KUKA KRL program: wkz6_off_st600.src, wkz6_off_st600.dat

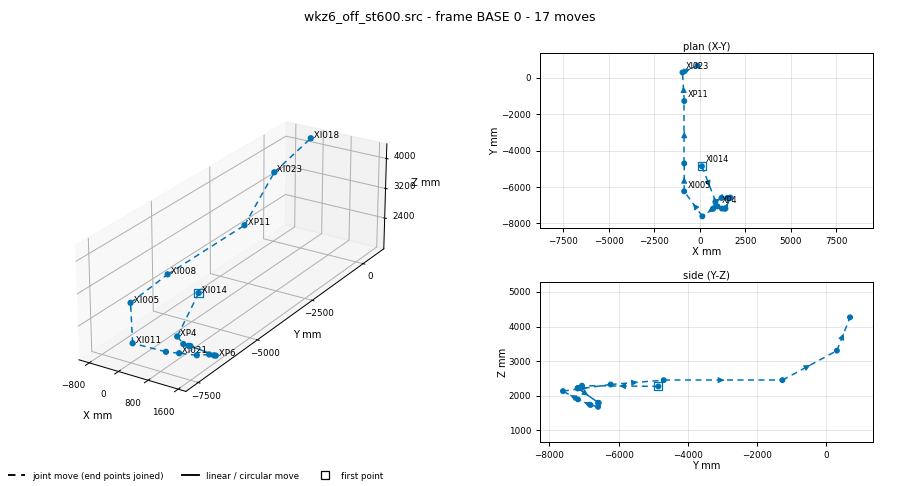
[picture p0: tool path of wkz6_off_st600.src in frame BASE 0, 17 of 17 moves have a stored position in this frame; points joined in program order, loops and branches not executed]
--- wkz6_off_st600.src ---
&ACCESS RVO4
&REL 118
&COMMENT Pega GRP AXOR GeoBox
&PARAM DISKPATH = KRC:\R1\Program\olp
&PARAM TEMPLATE = C:\KRC\Roboter\Template\vorgabe
&PARAM EDITMASK = *
DEF wkz6_off_st600( )
;FOLD INI
  ;FOLD BASISTECH INI
    GLOBAL INTERRUPT DECL 3 WHEN $STOPMESS==TRUE DO IR_STOPM ( )
    INTERRUPT ON 3
    BAS (#INITMOV,0)
  ;ENDFOLD (BASISTECH INI)
;FOLD GRIPPERTECH INI
USER_GRP(0,DUMMY,DUMMY,GDEFAULT)
;ENDFOLD (GRIPPERTECH INI)
  ;FOLD USER INI
    ;Make your modifications here

  ;ENDFOLD (USER INI)
;ENDFOLD (INI)

; Caracterizacao dos meios de producao
; Changes: Pega Gripper Axor na GeoBox
; Versao Atual: 20/08/2015
; Name: P13.050-R3

chk_w8_wechs_ok ( )   ; CHECK TOOL CHANGE

;FOLD ; Ponto Externo 7;%{PE}%R 8.2.20,%MKUKATPBASIS,%CCOMMENT,%VNORMAL,%P 2:Ponto Externo 7
;ENDFOLD
;FOLD PTP l014 Vel=100 % P_OLP34 Tool[8]:Tool Changer Base[0];%{PE}%R 8.2.20,%MKUKATPBASIS,%CMOVE,%VPTP,%P 1:PTP, 2:l014, 3:, 5:100, 7:P_OLP34
$BWDSTART=FALSE
PDAT_ACT=PP_OLP34
FDAT_ACT=Fl014
BAS(#PTP_PARAMS,100)
PTP Xl014
;ENDFOLD

; AGUARDA LIBERACAO PARA SAIR COM GARRA
;FOLD OUT 3378 'Lib. p/ retirar Gripper GeoBox' State=TRUE ;%{PE}%R 8.2.20,%MKUKATPBASIS,%COUT,%VOUTX,%P 2:3378, 3:Lib. p/ retirar Gripper GeoBox, 5:TRUE, 6:
$OUT[3378]=TRUE
;ENDFOLD
;FOLD WAIT FOR ( IN 3378 'Lib. p/ retirar Gripper GeoBox' );%{PE}%R 8.2.20,%MKUKATPBASIS,%CEXT_WAIT_FOR,%VEXT_WAIT_FOR,%P 2:, 4:, 5:$IN, 6:3378, 7:Lib. p/ retirar Gripper GeoBox, 9:
WAIT FOR  ( $IN[3378] )
;ENDFOLD
;FOLD OUT 3378 'Lib. p/ retirar Gripper GeoBox' State=FALSE ;%{PE}%R 8.2.20,%MKUKATPBASIS,%COUT,%VOUTX,%P 2:3378, 3:Lib. p/ retirar Gripper GeoBox, 5:FALSE, 6:
$OUT[3378]=FALSE
;ENDFOLD
;FOLD OUT 3348 'Fora area GEOBOX' State=FALSE ;%{PE}%R 8.2.20,%MKUKATPBASIS,%COUT,%VOUTX,%P 2:3348, 3:Fora area GEOBOX, 5:FALSE, 6:
$OUT[3348]=FALSE
;ENDFOLD

; LIGA INTERTRAVAMENTO 1 C/ R1 GARRA
;FOLD Collision.Monitoring_1_On ;%{PE}%MKUKATPUSER
COLLSTOP( 1, 1 ) ;Interrupt-Controlled
;ENDFOLD

; LIGA INTERTRAVAMENTO 5 C/ R5 GARRA
;FOLD Collision.Monitoring_5_On ;%{PE}%MKUKATPUSER
COLLSTOP( 5, 1 ) ;not Interrupt-Controlled
;ENDFOLD

;FOLD PTP P4 CONT Vel=100 % PDAT2 Tool[6]:Gripper G0100R Base[0];%{PE}%R 8.2.20,%MKUKATPBASIS,%CMOVE,%VPTP,%P 1:PTP, 2:P4, 3:C_DIS, 5:100, 7:PDAT2
$BWDSTART=FALSE
PDAT_ACT=PPDAT2
FDAT_ACT=FP4
BAS(#PTP_PARAMS,100)
PTP XP4 C_DIS
;ENDFOLD
;FOLD PTP P7 CONT Vel=100 % PDAT3 Tool[6]:Gripper G0100R Base[0];%{PE}%R 8.2.20,%MKUKATPBASIS,%CMOVE,%VPTP,%P 1:PTP, 2:P7, 3:C_DIS, 5:100, 7:PDAT3
$BWDSTART=FALSE
PDAT_ACT=PPDAT3
FDAT_ACT=FP7
BAS(#PTP_PARAMS,100)
PTP XP7 C_DIS
;ENDFOLD
;FOLD LIN l041 Vel=0.25 m/s L_OLP3 Tool[8]:Tool Changer Base[0];%{PE}%R 8.2.20,%MKUKATPBASIS,%CMOVE,%VLIN,%P 1:LIN, 2:l041, 3:, 5:0.25, 7:L_OLP3
$BWDSTART=FALSE
LDAT_ACT=LL_OLP3
FDAT_ACT=Fl041
BAS(#CP_PARAMS,0.25)
LIN Xl041
;ENDFOLD

; AGUARDA MPS DESTRAVADO
;FOLD OUT 224 'Bloquear MPS' State=FALSE ;%{PE}%R 8.2.20,%MKUKATPBASIS,%COUT,%VOUTX,%P 2:224, 3:Bloquear MPS, 5:FALSE, 6:
$OUT[224]=FALSE
;ENDFOLD
;FOLD OUT 223 'Desbloquear MPS' State=TRUE ;%{PE}%R 8.2.20,%MKUKATPBASIS,%COUT,%VOUTX,%P 2:223, 3:Desbloquear MPS, 5:TRUE, 6:
$OUT[223]=TRUE
;ENDFOLD
;FOLD WAIT FOR ( IN 217 'MPS Destravado' );%{PE}%R 8.2.20,%MKUKATPBASIS,%CEXT_WAIT_FOR,%VEXT_WAIT_FOR,%P 2:, 4:, 5:$IN, 6:217, 7:MPS Destravado, 9:
WAIT FOR  ( $IN[217] )
;ENDFOLD
;FOLD WAIT FOR NOT ( IN 221 'MPS Travado' );%{PE}%R 8.2.20,%MKUKATPBASIS,%CEXT_WAIT_FOR,%VEXT_WAIT_FOR,%P 2:NOT, 4:, 5:$IN, 6:221, 7:MPS Travado, 9:
WAIT FOR  NOT ( $IN[221] )
;ENDFOLD

;FOLD ; Posicao de Pega Gripper AXOR na GeoBox;%{PE}%R 8.2.20,%MKUKATPBASIS,%CCOMMENT,%VNORMAL,%P 2:Posicao de Pega Gripper AXOR  na  GeoBox
;ENDFOLD
;FOLD LIN P_DE11 Vel=0.25 m/s L_OLP4 Tool[8]:Tool Changer Base[0];%{PE}%R 8.2.20,%MKUKATPBASIS,%CMOVE,%VLIN,%P 1:LIN, 2:P_DE11, 3:, 5:0.25, 7:L_OLP4
$BWDSTART=FALSE
LDAT_ACT=LL_OLP4
FDAT_ACT=FP_DE11
BAS(#CP_PARAMS,0.25)
LIN XP_DE11
;ENDFOLD

;FOLD OUT 3379 'Lib. p/ sair c/ Gripper GeoBox' State=TRUE ;%{PE}%R 8.2.20,%MKUKATPBASIS,%COUT,%VOUTX,%P 2:3379, 3:Lib. p/ sair c/ Gripper GeoBox, 5:TRUE, 6:
$OUT[3379]=TRUE
;ENDFOLD

;FOLD WAIT FOR ( IN 219 'Posicao p/ Acoplamento OK' );%{PE}%R 8.2.20,%MKUKATPBASIS,%CEXT_WAIT_FOR,%VEXT_WAIT_FOR,%P 2:, 4:, 5:$IN, 6:219, 7:Posicao p/ Acoplamento OK, 9:
WAIT FOR  ( $IN[219] )
;ENDFOLD
;FOLD WAIT Time=0.5 sec;%{PE}%R 8.2.20,%MKUKATPBASIS,%CWAIT,%VWAIT,%P 3:0.5
WAIT SEC 0.5
;ENDFOLD
;FOLD OUT 223 'Desbloquear MPS' State=FALSE ;%{PE}%R 8.2.20,%MKUKATPBASIS,%COUT,%VOUTX,%P 2:223, 3:Desbloquear MPS, 5:FALSE, 6:
$OUT[223]=FALSE
;ENDFOLD
;FOLD OUT 224 'Bloquear MPS' State=TRUE ;%{PE}%R 8.2.20,%MKUKATPBASIS,%COUT,%VOUTX,%P 2:224, 3:Bloquear MPS, 5:TRUE, 6:
$OUT[224]=TRUE
;ENDFOLD
;FOLD WAIT FOR NOT ( IN 217 'MPS Destravado' );%{PE}%R 8.2.20,%MKUKATPBASIS,%CEXT_WAIT_FOR,%VEXT_WAIT_FOR,%P 2:NOT, 4:, 5:$IN, 6:217, 7:MPS Destravado, 9:
WAIT FOR  NOT ( $IN[217] )
;ENDFOLD
;FOLD WAIT FOR ( IN 221 'MPS Travado' );%{PE}%R 8.2.20,%MKUKATPBASIS,%CEXT_WAIT_FOR,%VEXT_WAIT_FOR,%P 2:, 4:, 5:$IN, 6:221, 7:MPS Travado, 9:
WAIT FOR  ( $IN[221] )
;ENDFOLD
;FOLD IBUS ON SEGMENT_4;%{PE}%R 8.2.20,%MKUKATPBASIS,%CIBUS,%VMAP,%P 2:#ON, 3:4
$IBUS_ON=IBUS_SEGMENT[4]
$IBUS_OFF=0
;ENDFOLD
;FOLD WAIT Time=0.5 sec;%{PE}%R 8.2.20,%MKUKATPBASIS,%CWAIT,%VWAIT,%P 3:0.5
WAIT SEC 0.5
;ENDFOLD

; ABRE GRAMPOS
;FOLD SET Z2.1 RPS AXOR State=OPN GDAT15;%{PE}%R 8.2.1,%MKUKATPGRP,%CGRP,%VGRP,%P 2:10, 4:1, 5:#NO, 6:GDAT15, 8:0, 10:0
H50(GRP,10,1,GGDAT15)
;ENDFOLD
;FOLD SET Z4.1 GRP AXOR State=OPN GDAT12;%{PE}%R 8.2.1,%MKUKATPGRP,%CGRP,%VGRP,%P 2:12, 4:1, 5:#NO, 6:GDAT12, 8:0, 10:0
H50(GRP,12,1,GGDAT12)
;ENDFOLD
;FOLD SET Z5.1/2/3/4 GRP AXOR State=OPN GDAT16;%{PE}%R 8.2.1,%MKUKATPGRP,%CGRP,%VGRP,%P 2:13, 4:1, 5:#NO, 6:GDAT16, 8:0, 10:0
H50(GRP,13,1,GGDAT16)
;ENDFOLD
;FOLD SET Z6.1/2/3/4 GRP AXOR State=OPN GDAT17;%{PE}%R 8.2.1,%MKUKATPGRP,%CGRP,%VGRP,%P 2:14, 4:1, 5:#NO, 6:GDAT17, 8:0, 10:0
H50(GRP,14,1,GGDAT17)
;ENDFOLD
;FOLD SET Z7.1/2 GRP AXOR State=OPN GDAT18;%{PE}%R 8.2.1,%MKUKATPGRP,%CGRP,%VGRP,%P 2:15, 4:1, 5:#NO, 6:GDAT18, 8:0, 10:0
H50(GRP,15,1,GGDAT18)
;ENDFOLD

; VERIFICA GRAMPOS ABERTOS
chk_w6_rps2_opn( )
chk_w6_grp4_opn( )
chk_w6_grp5_opn( )

; ABRE GRAMPO Z3.1 e VERIFICA
;FOLD SET Z3.1 GRP AXOR State=OPN GDAT13;%{PE}%R 8.2.1,%MKUKATPGRP,%CGRP,%VGRP,%P 2:11, 4:1, 5:#NO, 6:GDAT13, 8:0, 10:0
H50(GRP,11,1,GGDAT13)
;ENDFOLD
chk_w6_grp6_opn( )
chk_w6_grp7_opn( )
chk_w6_grp3_opn( )

; AGUARDA LIBERACAO PARA SAIR COM GARRA
;FOLD OUT 3379 'Lib. p/ sair c/ Gripper GeoBox' State=TRUE ;%{PE}%R 8.2.20,%MKUKATPBASIS,%COUT,%VOUTX,%P 2:3379, 3:Lib. p/ sair c/ Gripper GeoBox, 5:TRUE, 6:
$OUT[3379]=TRUE
;ENDFOLD
;FOLD WAIT FOR ( IN 3379 'Lib. p/ sair c/ Gripper GeoBox' );%{PE}%R 8.2.20,%MKUKATPBASIS,%CEXT_WAIT_FOR,%VEXT_WAIT_FOR,%P 2:, 4:, 5:$IN, 6:3379, 7:Lib. p/ sair c/ Gripper GeoBox, 9:
WAIT FOR  ( $IN[3379] )
;ENDFOLD
;FOLD OUT 3379 'Lib. p/ sair c/ Gripper GeoBox' State=FALSE ;%{PE}%R 8.2.20,%MKUKATPBASIS,%COUT,%VOUTX,%P 2:3379, 3:Lib. p/ sair c/ Gripper GeoBox, 5:FALSE, 6:
$OUT[3379]=FALSE
;ENDFOLD

;FOLD LIN P6 Vel=0.1 m/s CPDAT4 Tool[6]:Gripper G0100R Base[0];%{PE}%R 8.2.20,%MKUKATPBASIS,%CMOVE,%VLIN,%P 1:LIN, 2:P6, 3:, 5:0.1, 7:CPDAT4
$BWDSTART=FALSE
LDAT_ACT=LCPDAT4
FDAT_ACT=FP6
BAS(#CP_PARAMS,0.1)
LIN XP6
;ENDFOLD

;FOLD WAIT FOR ( IN 219 'Posicao p/ Acoplamento OK' ) CONT;%{PE}%R 8.2.20,%MKUKATPBASIS,%CEXT_WAIT_FOR,%VEXT_WAIT_FOR,%P 2:, 4:, 5:$IN, 6:219, 7:Posicao p/ Acoplamento OK, 9:CONTINUE
CONTINUE
WAIT FOR  ( $IN[219] )
;ENDFOLD

;FOLD PTP l036 CONT Vel=100 % P_OLP13 Tool[6]:Gripper G0100R Base[0];%{PE}%R 8.2.20,%MKUKATPBASIS,%CMOVE,%VPTP,%P 1:PTP, 2:l036, 3:C_DIS, 5:100, 7:P_OLP13
$BWDSTART=FALSE
PDAT_ACT=PP_OLP13
FDAT_ACT=Fl036
BAS(#PTP_PARAMS,100)
PTP Xl036 C_DIS
;ENDFOLD
;FOLD PTP l031 CONT Vel=100 % P_OLP14 Tool[6]:Gripper G0100R Base[0];%{PE}%R 8.2.20,%MKUKATPBASIS,%CMOVE,%VPTP,%P 1:PTP, 2:l031, 3:C_DIS, 5:100, 7:P_OLP14
$BWDSTART=FALSE
PDAT_ACT=PP_OLP14
FDAT_ACT=Fl031
BAS(#PTP_PARAMS,100)
PTP Xl031 C_DIS
;ENDFOLD
;FOLD PTP l026 CONT Vel=100 % P_OLP15 Tool[6]:Gripper G0100R Base[0];%{PE}%R 8.2.20,%MKUKATPBASIS,%CMOVE,%VPTP,%P 1:PTP, 2:l026, 3:C_DIS, 5:100, 7:P_OLP15
$BWDSTART=FALSE
PDAT_ACT=PP_OLP15
FDAT_ACT=Fl026
BAS(#PTP_PARAMS,100)
PTP Xl026 C_DIS
;ENDFOLD
;FOLD PTP l021 CONT Vel=100 % P_OLP16 Tool[6]:Gripper G0100R Base[0];%{PE}%R 8.2.20,%MKUKATPBASIS,%CMOVE,%VPTP,%P 1:PTP, 2:l021, 3:C_DIS, 5:100, 7:P_OLP16
$BWDSTART=FALSE
PDAT_ACT=PP_OLP16
FDAT_ACT=Fl021
BAS(#PTP_PARAMS,100)
PTP Xl021 C_DIS
;ENDFOLD

;FOLD PULSE 3335 'R3 retirou garra da Geo' State=TRUE Time=3 sec;%{PE}%R 8.2.20,%MKUKATPBASIS,%COUT,%VPULSE,%P 2:3335, 3:R3 retirou garra da Geo, 5:TRUE, 6:, 8:3
PULSE($OUT[3335], TRUE,3)
;ENDFOLD
;FOLD OUT 3348 'Fora area GEOBOX' State=TRUE ;%{PE}%R 8.2.20,%MKUKATPBASIS,%COUT,%VOUTX,%P 2:3348, 3:Fora area GEOBOX, 5:TRUE, 6:
$OUT[3348]=TRUE
;ENDFOLD

;FOLD PTP l016 Vel=100 % P_OLP17 Tool[6]:Gripper G0100R Base[0];%{PE}%R 8.2.20,%MKUKATPBASIS,%CMOVE,%VPTP,%P 1:PTP, 2:l016, 3:, 5:100, 7:P_OLP17
$BWDSTART=FALSE
PDAT_ACT=PP_OLP17
FDAT_ACT=Fl016
BAS(#PTP_PARAMS,100)
PTP Xl016
;ENDFOLD

; DESLIGA INTERTRAVAMENTO 5 C/ R5 GARRA
;FOLD Collision.Monitoring_5_Off . ;%{PE}%MKUKATPUSER
COLLSTOP( 5, 2+0 )
;ENDFOLD

;FOLD PTP l011 CONT Vel=100 % P_OLP18 Tool[6]:Gripper G0100R Base[0];%{PE}%R 8.2.20,%MKUKATPBASIS,%CMOVE,%VPTP,%P 1:PTP, 2:l011, 3:C_DIS, 5:100, 7:P_OLP18
$BWDSTART=FALSE
PDAT_ACT=PP_OLP18
FDAT_ACT=Fl011
BAS(#PTP_PARAMS,100)
PTP Xl011 C_DIS
;ENDFOLD
;FOLD PTP l005 CONT Vel=100 % P_OLP2 Tool[6]:Gripper G0100R Base[0];%{PE}%R 8.2.20,%MKUKATPBASIS,%CMOVE,%VPTP,%P 1:PTP, 2:l005, 3:C_DIS, 5:100, 7:P_OLP2
$BWDSTART=FALSE
PDAT_ACT=PP_OLP2
FDAT_ACT=Fl005
BAS(#PTP_PARAMS,100)
PTP Xl005 C_DIS
;ENDFOLD
;FOLD PTP l008 Vel=100 % P_OLP29 Tool[6]:Gripper G0100R Base[0];%{PE}%R 8.2.20,%MKUKATPBASIS,%CMOVE,%VPTP,%P 1:PTP, 2:l008, 3:, 5:100, 7:P_OLP29
$BWDSTART=FALSE
PDAT_ACT=PP_OLP29
FDAT_ACT=Fl008
BAS(#PTP_PARAMS,100)
PTP Xl008
;ENDFOLD

; DESLIGA INTERTRAVAMENTO 1 C/ R1 GARRA
;FOLD Collision.Monitoring_1_Off . ;%{PE}%MKUKATPUSER
COLLSTOP( 1, 2+0 )
;ENDFOLD


;FOLD PTP P11 CONT Vel=100 % PDAT8 Tool[6]:Gripper G0100R Base[0];%{PE}%R 8.2.20,%MKUKATPBASIS,%CMOVE,%VPTP,%P 1:PTP, 2:P11, 3:C_DIS, 5:100, 7:PDAT8
$BWDSTART=FALSE
PDAT_ACT=PPDAT8
FDAT_ACT=FP11
BAS(#PTP_PARAMS,100)
PTP XP11 C_DIS
;ENDFOLD

; FECHA GRAMPOS P/ DEPOSITAR GRIPPER NO DOCKING
;FOLD SET Z2.1 RPS AXOR State=CLO CONT at START Delay=1 ms;%{PE}%R 8.2.1,%MKUKATPGRP,%CGRP,%VGRP,%P 2:10, 4:2, 5:#YES, 6:GDAT1, 8:0, 10:1
TRIGGER WHEN DISTANCE=0 DELAY=1 DO H50(GRP_APO,10,2,GCONT) PRIO=-1
;ENDFOLD
;FOLD SET Z3.1 GRP AXOR State=CLO CONT at START Delay=1 ms;%{PE}%R 8.2.1,%MKUKATPGRP,%CGRP,%VGRP,%P 2:11, 4:2, 5:#YES, 6:GDAT1, 8:0, 10:1
TRIGGER WHEN DISTANCE=0 DELAY=1 DO H50(GRP_APO,11,2,GCONT) PRIO=-1
;ENDFOLD
;FOLD SET Z4.1 GRP AXOR State=CLO CONT at START Delay=1 ms;%{PE}%R 8.2.1,%MKUKATPGRP,%CGRP,%VGRP,%P 2:12, 4:2, 5:#YES, 6:GDAT1, 8:0, 10:1
TRIGGER WHEN DISTANCE=0 DELAY=1 DO H50(GRP_APO,12,2,GCONT) PRIO=-1
;ENDFOLD
;FOLD SET Z5.1/2/3/4 GRP AXOR State=CLO CONT at START Delay=1 ms;%{PE}%R 8.2.1,%MKUKATPGRP,%CGRP,%VGRP,%P 2:13, 4:2, 5:#YES, 6:GDAT1, 8:0, 10:1
TRIGGER WHEN DISTANCE=0 DELAY=1 DO H50(GRP_APO,13,2,GCONT) PRIO=-1
;ENDFOLD
;FOLD SET Z6.1/2/3/4 GRP AXOR State=CLO CONT at START Delay=1 ms;%{PE}%R 8.2.1,%MKUKATPGRP,%CGRP,%VGRP,%P 2:14, 4:2, 5:#YES, 6:GDAT1, 8:0, 10:1
TRIGGER WHEN DISTANCE=0 DELAY=1 DO H50(GRP_APO,14,2,GCONT) PRIO=-1
;ENDFOLD
;FOLD SET Z7.1/2 GRP AXOR State=CLO CONT at START Delay=1 ms;%{PE}%R 8.2.1,%MKUKATPGRP,%CGRP,%VGRP,%P 2:15, 4:2, 5:#YES, 6:GDAT1, 8:0, 10:1
TRIGGER WHEN DISTANCE=0 DELAY=1 DO H50(GRP_APO,15,2,GCONT) PRIO=-1
;ENDFOLD

;FOLD PTP l023 CONT Vel=100 % P_OLP25 Tool[6]:Gripper G0100R Base[0];%{PE}%R 8.2.20,%MKUKATPBASIS,%CMOVE,%VPTP,%P 1:PTP, 2:l023, 3:C_DIS, 5:100, 7:P_OLP25
$BWDSTART=FALSE
PDAT_ACT=PP_OLP25
FDAT_ACT=Fl023
BAS(#PTP_PARAMS,100)
PTP Xl023 C_DIS
;ENDFOLD
;FOLD PTP l018 CONT Vel=100 % P_OLP26 Tool[6]:Gripper G0100R Base[0];%{PE}%R 8.2.20,%MKUKATPBASIS,%CMOVE,%VPTP,%P 1:PTP, 2:l018, 3:C_DIS, 5:100, 7:P_OLP26
$BWDSTART=FALSE
PDAT_ACT=PP_OLP26
FDAT_ACT=Fl018
BAS(#PTP_PARAMS,100)
PTP Xl018 C_DIS
;ENDFOLD

END

--- wkz6_off_st600.dat ---
&ACCESS RVO4
&REL 118
&COMMENT Pega GRP AXOR GeoBox
&PARAM DISKPATH = KRC:\R1\Program\olp
&PARAM TEMPLATE = C:\KRC\Roboter\Template\vorgabe
&PARAM EDITMASK = *
DEFDAT  wkz6_off_st600
;FOLD EXTERNAL DECLARATIONS;%{PE}%MKUKATPBASIS,%CEXT,%VCOMMON,%P
;FOLD GRIPPERTECH EXT
EXT  H50 (INT  :IN,INT  :IN,INT  :IN,GRP_TYP  :IN )
;ENDFOLD (GRIPPERTECH EXT)
;FOLD SPOTTECH EXT

;ENDFOLD (SPOTTECH EXT)
;FOLD BASISTECH EXT;%{PE}%MKUKATPBASIS,%CEXT,%VEXT,%P
EXT  BAS (BAS_COMMAND  :IN,REAL  :IN )
DECL INT SUCCESS
;ENDFOLD (BASISTECH EXT)
;FOLD USER EXT;%{E}%MKUKATPUSER,%CEXT,%VEXT,%P
;Make your modifications here

;ENDFOLD (USER EXT)
;ENDFOLD (EXTERNAL DECLARATIONS)
DECL FDAT Fl005={TOOL_NO 6,BASE_NO 0,IPO_FRAME #BASE,POINT2[] " ",TQ_STATE FALSE}
DECL PDAT PP_OLP2={VEL 100.0,ACC 100.0,APO_DIST 100.0,APO_MODE #CDIS}
DECL E6POS Xl005={X -868.703979,Y -6232.00879,Z 2326.948,A 0.0,B 90.0,C -144.999695,S 2,T 35,E1 4350.0,E2 0.0,E3 0.0,E4 0.0,E5 0.0,E6 0.0}
DECL BASIS_SUGG_T LAST_BASIS={POINT1[] "P0                      ",POINT2[] "P0                      ",CP_PARAMS[] "CPDAT0                  ",PTP_PARAMS[] "PDAT0                   ",CONT[] "                        ",CP_VEL[] "2.0                     ",PTP_VEL[] " 100                    ",SYNC_PARAMS[] "SYNCDAT                 ",SPL_NAME[] "S0                      "}
DECL PDAT PPDAT2={VEL 100.0,ACC 100.0,APO_DIST 100.0,APO_MODE #CDIS}
DECL E6POS XP4={X 965.776001,Y -7059.44189,Z 2292.1189,A -54.9305382,B -71.0292969,C -129.947205,S 6,T 51,E1 5619.95313,E2 0.0,E3 0.0,E4 0.0,E5 0.0,E6 0.0}
DECL FDAT FP4={TOOL_NO 8,BASE_NO 0,IPO_FRAME #BASE,POINT2[] " ",TQ_STATE FALSE}
DECL LDAT LL_OLP3={VEL 0.25,ACC 100.0,APO_DIST 0.0,APO_FAC 0.0,ORI_TYP #VAR,CIRC_TYP #BASE,JERK_FAC 50.0}
DECL E6POS Xl041={X 1348.75903,Y -7181.64307,Z 2212.91699,A -90.0764694,B -74.8903122,C -89.8936768,S 6,T 51,E1 5699.86377,E2 0.0,E3 0.0,E4 0.0,E5 0.0,E6 0.0}
DECL FDAT Fl041={TOOL_NO 8,BASE_NO 0,IPO_FRAME #BASE,POINT2[] " "}
DECL LDAT LL_OLP4={VEL 0.25,ACC 100.0,APO_DIST 0.0,APO_FAC 0.0,ORI_TYP #VAR,CIRC_TYP #BASE,JERK_FAC 50.0}
DECL E6POS XP_DE11={X 1395.98999,Y -7181.66602,Z 2220.26611,A -88.7058029,B -74.86866,C -91.2107925,S 6,T 51,E1 5699.99805,E2 0.0,E3 0.0,E4 0.0,E5 0.0,E6 0.0}
DECL FDAT FP_DE11={TOOL_NO 8,BASE_NO 0,IPO_FRAME #BASE,POINT2[] " ",TQ_STATE FALSE}
DECL LDAT LCPDAT4={VEL 2.0,ACC 100.0,APO_DIST 100.0,APO_FAC 50.0,AXIS_VEL 100.0,AXIS_ACC 100.0,ORI_TYP #VAR,CIRC_TYP #BASE,JERK_FAC 50.0,GEAR_JERK 50.0,EXAX_IGN 0}
DECL E6POS XP6={X 1678.87805,Y -6580.3291,Z 1798.76196,A -108.197998,B -89.8673096,C 3.226717,S 6,T 51,E1 5699.99805,E2 0.0,E3 0.0,E4 0.0,E5 0.0,E6 0.0}
DECL FDAT FP6={TOOL_NO 6,BASE_NO 0,IPO_FRAME #BASE,POINT2[] " ",TQ_STATE FALSE}
DECL PDAT PP_OLP13={VEL 100.0,ACC 100.0,APO_DIST 30.0,APO_MODE #CDIS}
DECL E6POS Xl036={X 1631.401,Y -6588.33008,Z 1797.354,A 71.354332,B -89.986618,C -176.3564,S 6,T 51,E1 5700.0,E2 0.0,E3 0.0,E4 0.0,E5 0.0,E6 0.0}
DECL FDAT Fl036={TOOL_NO 6,BASE_NO 0,IPO_FRAME #BASE,POINT2[] " "}
DECL PDAT PP_OLP14={VEL 100.0,ACC 100.0,APO_DIST 30.0,APO_MODE #CDIS}
DECL E6POS Xl031={X 1506.66797,Y -6587.13916,Z 1785.50696,A 0.0,B -90.0,C -105.000099,S 6,T 51,E1 5700.0,E2 0.0,E3 0.0,E4 0.0,E5 0.0,E6 0.0}
DECL FDAT Fl031={TOOL_NO 6,BASE_NO 0,IPO_FRAME #BASE,POINT2[] " "}
DECL PDAT PP_OLP15={VEL 100.0,ACC 100.0,APO_DIST 30.0,APO_MODE #CDIS}
DECL E6POS Xl026={X 1179.49805,Y -6594.77002,Z 1681.64795,A 3.22912086E-07,B -80.0,C -105.000099,S 6,T 51,E1 5700.0,E2 0.0,E3 0.0,E4 0.0,E5 0.0,E6 0.0}
DECL FDAT Fl026={TOOL_NO 6,BASE_NO 0,IPO_FRAME #BASE,POINT2[] " "}
DECL PDAT PP_OLP16={VEL 100.0,ACC 100.0,APO_DIST 30.0,APO_MODE #CDIS}
DECL E6POS Xl021={X 846.315002,Y -6812.59424,Z 1735.85303,A -10.0776997,B -75.1255035,C -110.035896,S 6,T 51,E1 5400.0,E2 0.0,E3 0.0,E4 0.0,E5 0.0,E6 0.0}
DECL FDAT Fl021={TOOL_NO 6,BASE_NO 0,IPO_FRAME #BASE,POINT2[] " "}
DECL PDAT PP_OLP17={VEL 100.0,ACC 100.0,APO_DIST 100.0,APO_MODE #CDIS}
DECL E6POS Xl016={X 733.569397,Y -7176.80176,Z 1897.93896,A -168.100006,B -87.8154602,C 20.3269196,S 6,T 51,E1 5000.0,E2 0.0,E3 0.0,E4 0.0,E5 0.0,E6 0.0}
DECL FDAT Fl016={TOOL_NO 6,BASE_NO 0,IPO_FRAME #BASE,POINT2[] " "}
DECL PDAT PP_OLP18={VEL 100.0,ACC 100.0,APO_DIST 100.0,APO_MODE #CDIS}
DECL E6POS Xl011={X 130.889603,Y -7607.95313,Z 2134.82397,A -55.5008392,B -84.718399,C -156.303894,S 2,T 35,E1 4847.99023,E2 0.0,E3 0.0,E4 0.0,E5 0.0,E6 0.0}
DECL FDAT Fl011={TOOL_NO 6,BASE_NO 0,IPO_FRAME #BASE,POINT2[] " "}
DECL E6POS XP7={X 1208.60596,Y -7181.56104,Z 2220.479,A -89.919342,B -74.9435425,C -90.0644531,S 6,T 51,E1 5699.41602,E2 0.0,E3 0.0,E4 0.0,E5 0.0,E6 0.0}
DECL FDAT FP7={TOOL_NO 8,BASE_NO 0,IPO_FRAME #BASE,POINT2[] " ",TQ_STATE FALSE}
DECL PDAT PPDAT3={VEL 100.0,ACC 100.0,APO_DIST 100.0,APO_MODE #CDIS}
DECL PDAT PP_OLP25={VEL 100.0,ACC 100.0,APO_DIST 100.0,APO_MODE #CDIS}
DECL E6POS Xl023={X -961.385498,Y 300.348907,Z 3303.58203,A -88.2077789,B 5.06220913,C 129.177795,S 2,T 35,E1 -406.15509,E2 0.0,E3 0.0,E4 0.0,E5 0.0,E6 0.0}
DECL FDAT Fl023={TOOL_NO 6,BASE_NO 0,IPO_FRAME #BASE,POINT2[] " ",TQ_STATE FALSE}
DECL PDAT PP_OLP26={VEL 100.0,ACC 100.0,APO_DIST 100.0,APO_MODE #CDIS}
DECL E6POS Xl018={X -135.161301,Y 679.828918,Z 4266.34424,A 53.039341,B 47.648571,C 44.9270096,S 2,T 34,E1 -406.154602,E2 0.0,E3 0.0,E4 0.0,E5 0.0,E6 0.0}
DECL FDAT Fl018={TOOL_NO 6,BASE_NO 0,IPO_FRAME #BASE,POINT2[] " ",TQ_STATE FALSE}
DECL GRP_SUGG_T LAST_GRP={NUMBER[] "15                      ",STATE[] "2                       ",PARAMS[] "GDAT0                   "}
DECL GRP_TYP GGDAT15={G_APO #NO,GRP_TIME 0.200000003,CTRL #OFF,DLY 0,DST 1}
DECL GRP_TYP GGDAT8={G_APO #NO,GRP_TIME 0.200000003,CTRL #OFF,DLY 0,DST 1}
DECL GRP_TYP GGDAT16={G_APO #NO,GRP_TIME 0.200000003,CTRL #OFF,DLY 0,DST 1}
DECL GRP_TYP GGDAT17={G_APO #NO,GRP_TIME 0.200000003,CTRL #OFF,DLY 0,DST 1}
DECL GRP_TYP GGDAT18={G_APO #NO,GRP_TIME 0.200000003,CTRL #OFF,DLY 0,DST 1}
DECL GRP_TYP GGDAT9={G_APO #NO,GRP_TIME 0.200000003,CTRL #OFF,DLY 0,DST 1}
DECL GRP_TYP GGDAT10={G_APO #NO,GRP_TIME 0.200000003,CTRL #OFF,DLY 0,DST 1}
DECL E6POS XP11={X -864.721313,Y -1272.25403,Z 2452.09399,A 155.063095,B 89.9374084,C 10.21173,S 2,T 35,E1 -406.154388,E2 0.0,E3 0.0,E4 0.0,E5 0.0,E6 0.0}
DECL FDAT FP11={TOOL_NO 6,BASE_NO 0,IPO_FRAME #BASE,POINT2[] " ",TQ_STATE FALSE}
DECL PDAT PPDAT8={VEL 100.0,ACC 100.0,APO_DIST 100.0,APO_MODE #CDIS}
DECL PDAT PP_OLP29={VEL 100.0,ACC 100.0,APO_DIST 10.0,APO_MODE #CDIS}
DECL E6POS Xl008={X -864.721313,Y -4699.20508,Z 2452.09399,A 155.063095,B 89.9374084,C 10.21175,S 2,T 35,E1 3020.79712,E2 0.0,E3 0.0,E4 0.0,E5 0.0,E6 0.0}
DECL FDAT Fl008={TOOL_NO 6,BASE_NO 0,IPO_FRAME #BASE,POINT2[] " ",TQ_STATE FALSE}
DECL PDAT PP_OLP34={VEL 100.0,ACC 100.0,APO_DIST 10.0,APO_MODE #CDIS}
DECL E6POS Xl014={X 105.762299,Y -4854.60791,Z 2271.72192,A 91.3477173,B 9.41988564,C -178.989807,S 2,T 35,E1 3441.56201,E2 0.0,E3 0.0,E4 0.0,E5 0.0,E6 0.0}
DECL FDAT Fl014={TOOL_NO 8,BASE_NO 0,IPO_FRAME #BASE,POINT2[] " ",TQ_STATE FALSE}
DECL GRP_TYP GGDAT11={G_APO #NO,GRP_TIME 0.200000003,CTRL #OFF,DLY 0,DST 1}
DECL GRP_TYP GGDAT12={G_APO #NO,GRP_TIME 0.200000003,CTRL #OFF,DLY 0,DST 1}
DECL GRP_TYP GGDAT13={G_APO #NO,GRP_TIME 0.200000003,CTRL #OFF,DLY 0,DST 1}
DECL GRP_TYP GCONT={G_APO #YES,GRP_TIME 0.0,CTRL #OFF,DLY 0,DST 0}
DECL E6POS XP1={X 1393.849,Y -7181.67676,Z 2220.25,A -90.1178436,B -74.8756638,C -89.8492279,S 6,T 51,E1 5700.0,E2 0.0,E3 0.0,E4 0.0,E5 0.0,E6 0.0}
DECL FDAT FP1={TOOL_NO 8,BASE_NO 0,IPO_FRAME #BASE,POINT2[] " ",TQ_STATE FALSE}
DECL PDAT PPDAT1={VEL 100.0,ACC 100.0,APO_DIST 100.0}
ENDDAT
